FUNCTION_BLOCK FB_HTTP_Get_SmartMeter
VAR_INPUT
	bSend				: BOOL;
	timDataMomentan:REFERENCE TO ST_timData;
	nettoEffektWh:REFERENCE TO REAL;
END_VAR
VAR_IN_OUT
	fbClient			: FB_IotHttpClient;
END_VAR
VAR_OUTPUT
	bBusy				: BOOL;
	bError				: BOOL;
END_VAR
VAR
	fbRequest			: FB_IotHttpRequest;
	fbJson				: FB_JsonDomParser;
	
		fbJsonDataType	: FB_JsonReadWriteDataType;
		felkod			: HRESULT;			
	pContent: PVOID;
	nState				: UDINT;
	RisingEdge			: R_TRIG;
	
	bGetContentResult	: BOOL;
	sContent			: STRING(1100);
	
	bGetJsonResult		: BOOL;
	jsonDoc				: SJsonValue;
	jsonVal				: SJsonValue;
	sResultValue		: STRING;
	
	nReqCount			: UDINT;	
	nResCount			: UDINT;
	nValidResCount		: UDINT;
	nErrCount			: UDINT;
	Vaerde: LINT;
	

	SaaldEffektWh: REAL;
	KoeptEffektWh: REAL;

	Effektlaegsta: REAL :=100000.0 ;
	Effekthoegsta: REAL;
	NettoEnergiAccumulerat: REAL;
	SaaldEnergiAccumulerat: REAL;
	KoeptEnergiAccumulerat: REAL;

	Funkar: BOOL;
	nisse: INT;
	stSmartDataMomentan: SmartMeterValues;
END_VAR

RisingEdge(CLK:= bSend );



CASE nState OF
0:	
	IF RisingEdge.Q THEN 
		IF Funkar:= fbRequest.SendRequest(sUri:='/smartmeter/api/read', fbClient:=fbClient, eRequestType:=ETcIotHttpRequestType.HTTP_Get, 0, 0, 0) THEN				
		
		nState:= 1;
			nReqCount:= nReqCount+1;
			bBusy:= TRUE;
			bError:= FALSE;
		END_IF				
	END_IF
1:

	IF NOT fbRequest.bBusy THEN
		bError:= TRUE;
		IF NOT fbRequest.bError THEN	
			

			
//Hämta data från mätarens HTTP REST API och lägg i string
			bGetContentResult:= fbRequest.GetContent(pContent:= ADR(sContent), nContentSize:= SIZEOF(sContent), bSetNullTermination:= TRUE);
			
			
			IF fbRequest.nStatusCode >= 200 AND fbRequest.nStatusCode < 300 THEN
				bGetJsonResult:= FALSE;
			
			//Kopiera hela den importerade JSON-formaterade datasträngen och lägg i en motsvarande TwinCAT-struktur
			IF fbJsonDataType.SetSymbolFromJson(sContent, 'SmartMeterValues', SIZEOF(stSmartDataMomentan), ADR(stSmartDataMomentan), hrErrorCode=> felkod) THEN
						bError:= FALSE;
					END_IF	
			
			//räkna ut lägsta och högsta effekt
			IF felkod = 0 THEN
					
				//timDataMomentan.nettoEnergi := STRING_TO_REAL(stSmartDataMomentan.PowerDeliveredNetto);
				SaaldEffektWh:= STRING_TO_REAL(stSmartDataMomentan.PowerReturned_total);
				KoeptEffektWh := STRING_TO_REAL(stSmartDataMomentan.PowerDelivered_total);
				nettoEffektWh:= (KoeptEffektWh-SaaldEffektWh);
			END_IF	
			
				//skriv in i Struct
				timDataMomentan.nettoEnergi:= timDataMomentan.nettoEnergi+ (nettoEffektWh/144000);
				timDataMomentan.saaldEnergi:= timDataMomentan.saaldEnergi+ (SaaldEffektWh/144000);
				timDataMomentan.KoeptEnergi:= timDataMomentan.KoeptEnergi+(KoeptEffektWh/144000);
				
				
				IF timDataMomentan.laegstaNettoEffekt> nettoEffektWh/1000 THEN 	
					timDataMomentan.laegstaNettoEffekt:=nettoEffektWh/1000;
				ELSIF timDataMomentan.toppNettoEffekt< nettoEffektWh/1000 THEN 	
					timDataMomentan.toppNettoEffekt:=nettoEffektWh/1000;			
				END_IF
				
				
	

			
				nResCount:= nResCount+1;			
			END_IF
		END_IF
			nisse:=nisse+1;
		nState:= 2;
		bBusy:= FALSE;
		IF bError THEN
			nErrCount:= nErrCount+1;
		END_IF
	END_IF  	

2:   //Räkna ut pengar
timDataMomentan.saaltSolceller:= timDataMomentan.saaltSolceller+(SaaldEffektWh/144000*(timDataMomentan.timPris+GVL.NaetNyttaKWh+GVL.SkatteAvdragKWh));
timDataMomentan.Koept:= timDataMomentan.Koept + KoeptEffektWh/144000*(timDataMomentan.timPris+GVL.ElOeverfoeringsAvgiftEonKWh+GVL.EnergiskattKWh+GVL.MomsKWh+GVL.PaaslagMinusRabattKWh);


//IF timDataMomentan.husnettoEffekt

nState:= 0;

	
END_CASE

END_FUNCTION_BLOCK

(* stored: Version 1.1.0.1, ProductVersion 3.1.4024.12
   POU FB_HTTP_Get_SmartMeter: Id {10604ea1-d5d2-4f3e-b891-4dec4529946c}, SpecialFunc None *)
